Fanuc KAREL source: IO0224.KL

PROGRAM IO0224
%STACKSIZE=65535
%PRIORITY=65535
%NOLOCKGROUP
ROUTINE RTEST FROM IO0224
ROUTINE RTEST
VAR
L1 : ARRAY[3] OF INTEGER
L2 : XYZWPR
L3 : JOINTPOS9
L4 : POSITION
S1 : INTEGER
S2 : INTEGER
S3 : INTEGER
U2C_40 : BOOLEAN -- ASSUMED 2C source type; see uncertainty report
U2C_41 : INTEGER -- ASSUMED 2C source type; see uncertainty report
BEGIN
S1=1
L1[1]=2
U2C_40=TRUE
U2C_41=1065353216
SET_VAR(S3,'*SYSTEM*','$MNUTOOLNUM[1]',S1,S2)
END RTEST
BEGIN
RTEST
END IO0224
